// TIA Portal V18 export
DATA_BLOCK "04_SPEED"   // DB6, F_DB
{ S7_Optimized_Access := 'TRUE'; DB_Accessible_From_OPC_UA := 'FALSE' }
VERSION : 0.1
// stored: AutoNumber true, DBAccessibleFromOPCUA false, DBAccessibleFromWebserver true
   VAR
      AlwaysFALSE : Bool;
      AlwaysTRUE : Bool;
      "No Operation" : Bool;
      "Safety Encoder 0001 Sensor 1 Healthy [ =S1+PC1.CC1-X81001 ]" : Bool;
      "Safety Encoder 0002 Sensor 1 Healthy [ =S2+PC2.CC1-X81001 ]" : Bool;
      "Safety Encoder 0001 Sensor 2 Healthy [ =S1+PC1.CC1-X81001 ]" : Bool;
      "Safety Encoder 0002 Sensor 2 Healthy [ =S2+PC2.CC1-X81001 ]" : Bool;
      "Safety Encoder 0001 Healthy [ =S1+PC1.CC1-X81001 ]" : Bool;
      "Safety Encoder 0002 Healthy [ =S2+PC2.CC1-X81001 ]" : Bool;
   END_VAR
BEGIN
END_DATA_BLOCK
